// TIA Portal V18 export
DATA_BLOCK "DL_Vars"   // DB51051
{ S7_Optimized_Access := 'FALSE'; DB_Accessible_From_OPC_UA := 'FALSE' }
VERSION : 0.1
// stored: AutoNumber false, DBAccessibleFromOPCUA false, IsOnlyStoredInLoadMemory false, IsWriteProtectedInAS false
   VAR
      Vars { S7_SetPoint := 'True'} : "UDT_DL_Vars";
   END_VAR
BEGIN
END_DATA_BLOCK
